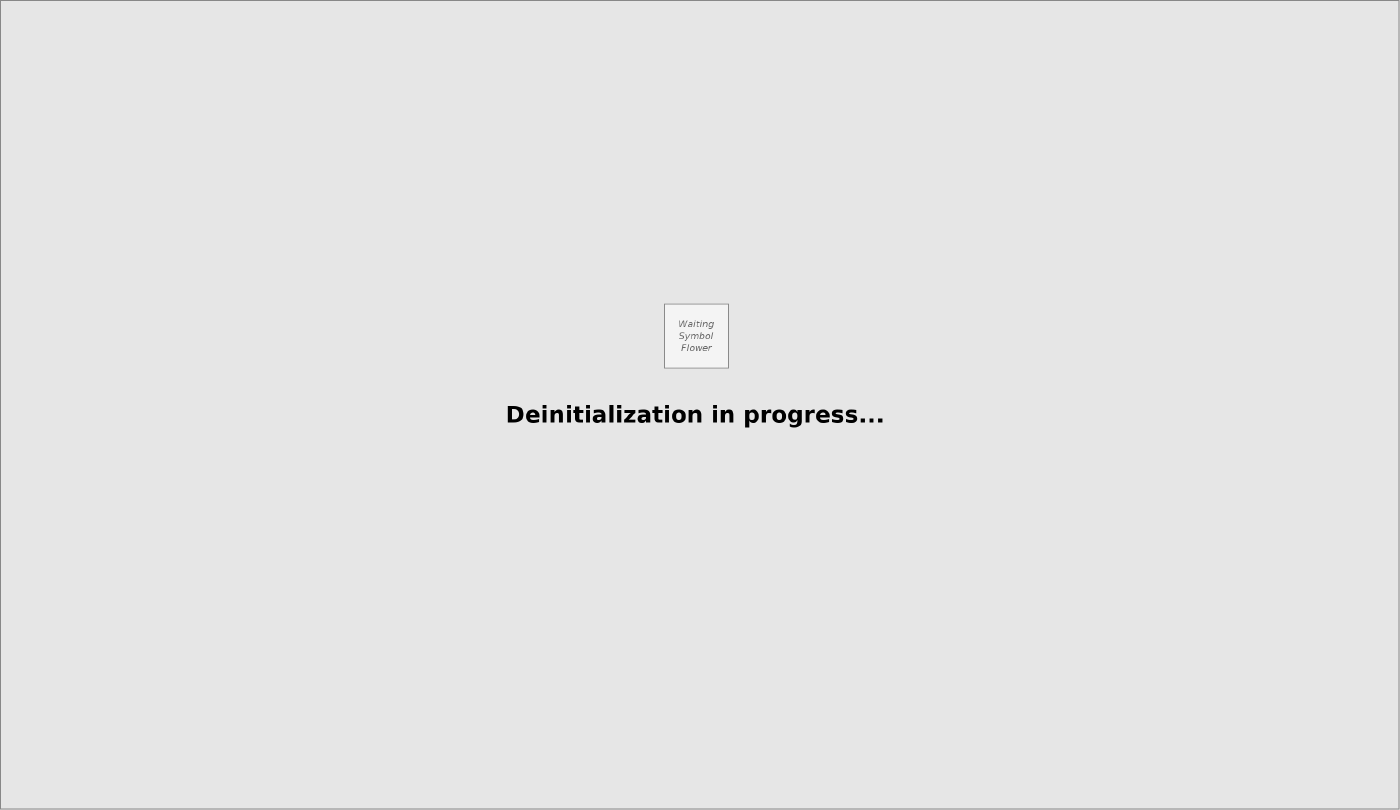
VISUALIZATION PageAborting  // 1520x880
    Group (530,330 450x140)
        WaitingSymbolFlower (191,0 70x70)
        Label (0,100 450x40), "Deinitialization in progress..."
END_VISUALIZATION

(* stored: Version 1.1.0.1, ProductVersion 3.1.4024.9
   Visu PageAborting: Id {e08dd844-e3f3-4755-be84-2500a3705f4f} *)
